TYPE
    ST_TestResult :
    STRUCT
        TestCompleted : BOOL;
        TestFailed    : BOOL;
        FailMessage   : T_MaxString;
    END_STRUCT
END_TYPE

(* stored: Version 1.1.0.1, ProductVersion 3.1.4024.11
   DUT ST_TestResult: Id {2865ee9b-7ea4-4a4a-a4e5-3044e35b8d34} *)
